# EPICS substitutions: motionSetPointsApp/Db/motionSetPointsSingleAxis.substitutions
file "$(TOP)/motionSetPointsApp/Db/motionSetPointsHeader.template" {
	pattern{ P, LOOKUP, COORD0 }
	{ "\$(P)", "\$(LOOKUP)", "0" }
}

file "$(TOP)/motionSetPointsApp/Db/single_axis.template" {
	pattern{ P, AXIS_NUM, AXIS, LOOKUP }
	{ "\$(P)", "0", "\$(AXIS1)", "\$(LOOKUP)" }
}
